FUNCTION_BLOCK CSV_WRITER_5 (* Service Interface Function Block Type *)
  (* Description: Copyright (c) 2012 ACIN This program and the accompanying materials are made available under the terms of the Eclipse Public License 2.0 which is available at https://www.eclipse.org/legal/epl-2.0/ SPDX-License-Identifier: EPL-2.0 *)
  (* Version 1.0, 2012-06-16, Alois Zoitl, ACIN *)
  (* Version 3.0, 2025-04-14, Patrick Aigner, changed package *)
  PACKAGE eclipse4diac::utils;
  {SET_ATTRIBUTE(eclipse4diac::core::GenericClassName, 'GEN_CSV_WRITER')}
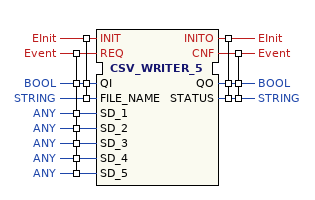
  EVENT_INPUT
    INIT : EInit WITH QI, FILE_NAME; (* Service Initialization *)
    REQ WITH QI, SD_1, SD_2, SD_3, SD_4, SD_5; (* Service Request *)
  END_EVENT
  EVENT_OUTPUT
    INITO : EInit WITH QO, STATUS; (* Initialization Confirm *)
    CNF WITH QO, STATUS; (* Confirmation of Requested Service *)
  END_EVENT
  VAR_INPUT
    QI : BOOL; (* Event Input Qualifier *)
    FILE_NAME : STRING; (* Service Parameters *)
    SD_1 : ANY; (* Output data to resource *)
    SD_2 : ANY;
    SD_3 : ANY;
    SD_4 : ANY;
    SD_5 : ANY;
  END_VAR
  VAR_OUTPUT
    QO : BOOL; (* Event Output Qualifier *)
    STATUS : STRING; (* File access status *)
  END_VAR
END_FUNCTION_BLOCK
